// TIA Portal V19 export
TYPE "LAF_typeEmInterface"
// Interface to control and monitor the EM from an HMI
// stored: Access Published
   STRUCT
      interlinkMode : "LUC_typeInterlinkMode";
      commands : "LAF_typeEmCommandsInterface";
      status { ExternalWritable := 'False'} : "LAF_typeEmStatus";
      alarms { ExternalWritable := 'False'} : "LAF_typeAlarms";
   END_STRUCT;
END_TYPE
